Universal Robots PolyScope program: house.urp

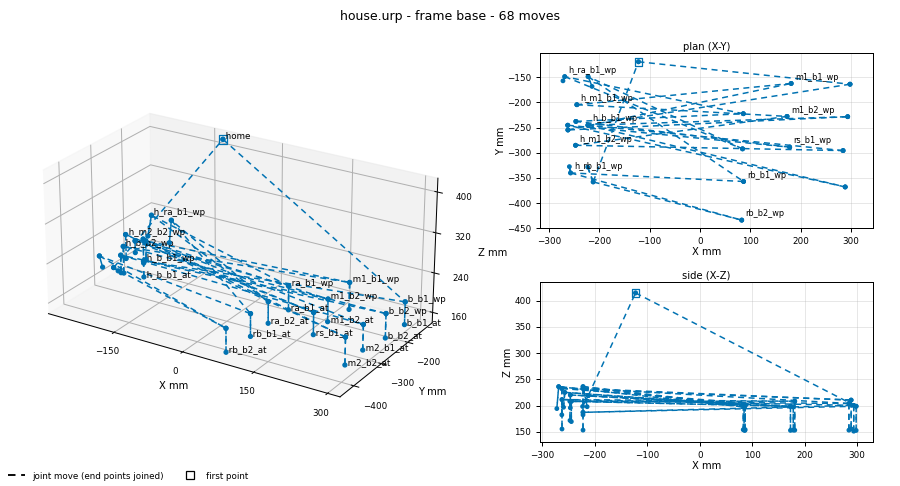
[picture p0: tool path of house.urp in frame base, 68 of 68 moves have a stored position in this frame; points joined in program order, loops and branches not executed]
Program house (installation=default directory=/programs/ITER createdIn=5.3.1.64192 lastSavedIn=5.3.1.64192 robotSerialNumber=20195300365)
Calibrated DH parameters: a=[-0.000093, -0.190649, -0.212673, 0.000091, -0.000205, 0]; d=[0.151591, 44.061648, -42.488068, -1.442789, 0.085322, 0.091911]; alpha=[1.570082, -0.003447, 0.007513, 1.572293, -1.571904, 0]; deltaTheta=[0, -0.672656, 0.728185, -0.055522, 0.000005, 0]
Robot Program (runOnlyOnce=true)
  URCap Gripper Activate (Robotiq_Grippers, Robotiq Inc.) dataModel(ResetAndActivateKey=false)
  URCap Gripper (Robotiq_Grippers, Robotiq Inc.) dataModel(position=50.0, force=100.0, speed=100.0, positionInDouble=50.0, forceInDouble=100.0, speedInDouble=100.0, slaveIds=[9], blocking=true)
  MoveJ speed 60 deg/s, acceleration 80 deg/s^2 (useActiveTCP=true) feature=Base
    Waypoint home: TCP in base x=-122.15 y=-119.32 z=414.454 mm, rx=2.2563 ry=2.1459 rz=-0.0481 rad; joints [-85.681, -56.776, -79.802, -131.025, 89.944, -262.833] deg
  Folder Base
    MoveJ speed 60 deg/s, acceleration 80 deg/s^2 (useActiveTCP=true) feature=Base
      Waypoint b_b1_wp: TCP in base x=297.989 y=-163.874 z=198.695 mm, rx=2.2416 ry=2.1933 rz=-0.0875 rad; joints [-5.657, -99.775, -108.03, -64.017, 87.69, -183.98] deg
      Waypoint b_b1_at: TCP in base x=297.98 y=-163.89 z=152.63 mm, rx=2.2418 ry=2.1932 rz=-0.0874 rad; joints [-5.678, -106.278, -114.473, -51.073, 87.63, -183.927] deg
      URCap Gripper (Robotiq_Grippers, Robotiq Inc.) dataModel(position=100.0, force=100.0, speed=100.0, positionInDouble=100.0, forceInDouble=100.0, speedInDouble=100.0, slaveIds=[9], blocking=true)
      Waypoint b_b1_wp: TCP in base x=297.989 y=-163.874 z=198.695 mm, rx=2.2416 ry=2.1933 rz=-0.0875 rad; joints [-5.657, -99.775, -108.03, -64.017, 87.69, -183.98] deg
      Waypoint h_b_b1_wp: TCP in base x=-222.187 y=-245.349 z=187.06 mm, rx=-3.1315 ry=0.0204 rz=0.0123 rad; joints [-108.957, -99.116, -113.081, -58.146, 89.665, -197.782] deg
      Waypoint h_b_b1_at: TCP in base x=-222.188 y=-245.348 z=153.24 mm, rx=-3.1314 ry=0.0204 rz=0.0122 rad; joints [-108.969, -104.391, -117.643, -48.312, 89.612, -197.745] deg
      URCap Gripper (Robotiq_Grippers, Robotiq Inc.) dataModel(position=50.0, force=100.0, speed=100.0, positionInDouble=50.0, forceInDouble=100.0, speedInDouble=100.0, slaveIds=[9], blocking=true)
      Waypoint h_b_b1_wp: TCP in base x=-222.187 y=-245.349 z=187.06 mm, rx=-3.1315 ry=0.0204 rz=0.0123 rad; joints [-108.957, -99.116, -113.081, -58.146, 89.665, -197.782] deg
    MoveJ speed 60 deg/s, acceleration 80 deg/s^2 (useActiveTCP=true) feature=Base
      Waypoint b_b2_wp: TCP in base x=293.357 y=-228.364 z=200.348 mm, rx=2.2516 ry=2.1757 rz=-0.0473 rad; joints [-17.02, -106.79, -99.111, -64.372, 88.479, -194.689] deg
      Waypoint b_b2_at: TCP in base x=293.371 y=-228.346 z=151.163 mm, rx=2.2516 ry=2.1757 rz=-0.0473 rad; joints [-17.033, -113.072, -105.562, -51.642, 88.423, -194.639] deg
      URCap Gripper (Robotiq_Grippers, Robotiq Inc.) dataModel(position=100.0, force=100.0, speed=100.0, positionInDouble=100.0, forceInDouble=100.0, speedInDouble=100.0, slaveIds=[9], blocking=true)
      Waypoint b_b2_wp: TCP in base x=293.357 y=-228.364 z=200.348 mm, rx=2.2516 ry=2.1757 rz=-0.0473 rad; joints [-17.02, -106.79, -99.111, -64.372, 88.479, -194.689] deg
      Waypoint h_b_b2_wp: TCP in base x=-262.196 y=-254.726 z=211.351 mm, rx=-3.0605 ry=0.0443 rz=-0.0223 rad; joints [-114.749, -105.359, -96.042, -73.109, 89.199, -202.734] deg
      Waypoint h_b_b2_at: TCP in base x=-262.208 y=-254.718 z=155.33 mm, rx=-3.0605 ry=0.0443 rz=-0.0223 rad; joints [-114.774, -111.736, -104.192, -58.581, 89.146, -202.674] deg
      URCap Gripper (Robotiq_Grippers, Robotiq Inc.) dataModel(position=50.0, force=100.0, speed=100.0, positionInDouble=50.0, forceInDouble=100.0, speedInDouble=100.0, slaveIds=[9], blocking=true)
      Waypoint h_b_b2_wp: TCP in base x=-262.196 y=-254.726 z=211.351 mm, rx=-3.0605 ry=0.0443 rz=-0.0223 rad; joints [-114.749, -105.359, -96.042, -73.109, 89.199, -202.734] deg
  Folder Mid_1
    MoveJ speed 60 deg/s, acceleration 80 deg/s^2 (useActiveTCP=true) feature=Base
      Waypoint m1_b1_wp: TCP in base x=181.055 y=-162.39 z=208.274 mm, rx=2.2824 ry=2.1481 rz=-0.0224 rad; joints [-9.334, -71.677, -131.429, -67.006, 89.476, -185.444] deg
      Waypoint m1_b1_at: TCP in base x=181.066 y=-162.388 z=153.109 mm, rx=2.2824 ry=2.1481 rz=-0.0224 rad; joints [-9.367, -82.083, -142.13, -45.899, 89.364, -185.356] deg
      URCap Gripper (Robotiq_Grippers, Robotiq Inc.) dataModel(position=100.0, force=100.0, speed=100.0, positionInDouble=100.0, forceInDouble=100.0, speedInDouble=100.0, slaveIds=[9], blocking=true)
      Waypoint m1_b1_wp: TCP in base x=181.055 y=-162.39 z=208.274 mm, rx=2.2824 ry=2.1481 rz=-0.0224 rad; joints [-9.334, -71.677, -131.429, -67.006, 89.476, -185.444] deg
      Waypoint h_m1_b1_wp: TCP in base x=-244.449 y=-204.582 z=208.1 mm, rx=2.2684 ry=2.1196 rz=0.0229 rad; joints [-116.825, -93.932, -112.747, -63.308, 92.582, -292.535] deg
      Waypoint h_m1_b1_at: TCP in base x=-244.447 y=-204.577 z=169.457 mm, rx=2.2685 ry=2.1196 rz=0.0229 rad; joints [-116.841, -99.299, -118.834, -51.852, 92.525, -292.487] deg
      URCap Gripper (Robotiq_Grippers, Robotiq Inc.) dataModel(position=50.0, force=100.0, speed=100.0, positionInDouble=50.0, forceInDouble=100.0, speedInDouble=100.0, slaveIds=[9], blocking=true)
      Waypoint h_m1_b1_wp: TCP in base x=-244.449 y=-204.582 z=208.1 mm, rx=2.2684 ry=2.1196 rz=0.0229 rad; joints [-116.825, -93.932, -112.747, -63.308, 92.582, -292.535] deg
    MoveJ speed 60 deg/s, acceleration 80 deg/s^2 (useActiveTCP=true) feature=Base
      Waypoint m1_b2_wp: TCP in base x=172.9 y=-227.784 z=198.59 mm, rx=2.2733 ry=2.1297 rz=0.0128 rad; joints [-25.861, -85.885, -124.428, -58.034, 90.195, -201.672] deg
      Waypoint m1_b2_at: TCP in base x=172.893 y=-227.779 z=152.722 mm, rx=2.2733 ry=2.1297 rz=0.0127 rad; joints [-25.879, -94.277, -131.683, -42.391, 90.103, -201.614] deg
      URCap Gripper (Robotiq_Grippers, Robotiq Inc.) dataModel(position=100.0, force=100.0, speed=100.0, positionInDouble=100.0, forceInDouble=100.0, speedInDouble=100.0, slaveIds=[9], blocking=true)
      Waypoint m1_b2_wp: TCP in base x=172.9 y=-227.784 z=198.59 mm, rx=2.2733 ry=2.1297 rz=0.0128 rad; joints [-25.861, -85.885, -124.428, -58.034, 90.195, -201.672] deg
      Waypoint h_m1_b2_wp: TCP in base x=-247.009 y=-285.144 z=208.116 mm, rx=2.2684 ry=2.1195 rz=0.0229 rad; joints [-111.389, -107.719, -95.772, -66.28, 92.556, -287.152] deg
      Waypoint h_m1_b2_at: TCP in base x=-246.994 y=-285.166 z=171.647 mm, rx=2.2684 ry=2.1196 rz=0.0229 rad; joints [-111.399, -111.783, -101.037, -56.949, 92.516, -287.113] deg
      URCap Gripper (Robotiq_Grippers, Robotiq Inc.) dataModel(position=50.0, force=100.0, speed=100.0, positionInDouble=50.0, forceInDouble=100.0, speedInDouble=100.0, slaveIds=[9], blocking=true)
      Waypoint h_m1_b2_wp: TCP in base x=-247.009 y=-285.144 z=208.116 mm, rx=2.2684 ry=2.1195 rz=0.0229 rad; joints [-111.389, -107.719, -95.772, -66.28, 92.556, -287.152] deg
  Folder Mid_2
    MoveJ speed 60 deg/s, acceleration 80 deg/s^2 (useActiveTCP=true) feature=Base
      Waypoint m2_b1_wp: TCP in base x=284.16 y=-295.685 z=203.947 mm, rx=2.2476 ry=2.1381 rz=-0.0269 rad; joints [-27.296, -114.823, -87.386, -65.934, 88.586, -204.141] deg
      Waypoint m2_b1_at: TCP in base x=284.146 y=-295.69 z=153.108 mm, rx=2.2477 ry=2.1381 rz=-0.0269 rad; joints [-27.314, -120.451, -93.885, -53.812, 88.539, -204.094] deg
      URCap Gripper (Robotiq_Grippers, Robotiq Inc.) dataModel(position=100.0, force=100.0, speed=100.0, positionInDouble=100.0, forceInDouble=100.0, speedInDouble=100.0, slaveIds=[9], blocking=true)
      Waypoint m2_b1_wp: TCP in base x=284.16 y=-295.685 z=203.947 mm, rx=2.2476 ry=2.1381 rz=-0.0269 rad; joints [-27.296, -114.823, -87.386, -65.934, 88.586, -204.141] deg
      Waypoint h_m2_b1_wp: TCP in base x=-222.193 y=-245.34 z=232.403 mm, rx=-3.1314 ry=0.0205 rz=0.0123 rad; joints [-108.936, -94.247, -105.13, -70.966, 89.712, -197.837] deg
      Waypoint h_m2_b1_at: TCP in base x=-222.194 y=-245.343 z=182.32 mm, rx=-3.1314 ry=0.0205 rz=0.0122 rad; joints [-108.96, -99.771, -113.792, -56.782, 89.658, -197.776] deg
      URCap Gripper (Robotiq_Grippers, Robotiq Inc.) dataModel(position=50.0, force=100.0, speed=100.0, positionInDouble=50.0, forceInDouble=100.0, speedInDouble=100.0, slaveIds=[9], blocking=true)
      Waypoint h_m2_b1_wp: TCP in base x=-222.193 y=-245.34 z=232.403 mm, rx=-3.1314 ry=0.0205 rz=0.0123 rad; joints [-108.936, -94.247, -105.13, -70.966, 89.712, -197.837] deg
    MoveJ speed 60 deg/s, acceleration 80 deg/s^2 (useActiveTCP=true) feature=Base
      Waypoint m2_b2_wp: TCP in base x=288.413 y=-367.875 z=210.448 mm, rx=2.2648 ry=2.1717 rz=-0.0293 rad; joints [-35.505, -129.071, -61.562, -79.296, 89.186, -212.92] deg
      Waypoint m2_b2_at: TCP in base x=288.4 y=-367.879 z=155.646 mm, rx=2.2649 ry=2.1717 rz=-0.0293 rad; joints [-35.528, -133.111, -69.75, -67.072, 89.162, -212.863] deg
      URCap Gripper (Robotiq_Grippers, Robotiq Inc.) dataModel(position=100.0, force=100.0, speed=100.0, positionInDouble=100.0, forceInDouble=100.0, speedInDouble=100.0, slaveIds=[9], blocking=true)
      Waypoint m2_b2_wp: TCP in base x=288.413 y=-367.875 z=210.448 mm, rx=2.2648 ry=2.1717 rz=-0.0293 rad; joints [-35.505, -129.071, -61.562, -79.296, 89.186, -212.92] deg
      Waypoint h_m2_b2_wp: TCP in base x=-262.568 y=-245.346 z=232.504 mm, rx=-3.1314 ry=0.0205 rz=0.0123 rad; joints [-115.613, -101.169, -97.08, -72.022, 89.654, -204.539] deg
      Waypoint h_m2_b2_at: TCP in base x=-262.563 y=-245.347 z=182.321 mm, rx=-3.1314 ry=0.0204 rz=0.0123 rad; joints [-115.635, -106.202, -105.428, -58.642, 89.608, -204.482] deg
      URCap Gripper (Robotiq_Grippers, Robotiq Inc.) dataModel(position=50.0, force=100.0, speed=100.0, positionInDouble=50.0, forceInDouble=100.0, speedInDouble=100.0, slaveIds=[9], blocking=true)
      Waypoint h_m2_b2_wp: TCP in base x=-262.568 y=-245.346 z=232.504 mm, rx=-3.1314 ry=0.0205 rz=0.0123 rad; joints [-115.613, -101.169, -97.08, -72.022, 89.654, -204.539] deg
  Folder Roof_Support
    MoveJ speed 60 deg/s, acceleration 80 deg/s^2 (useActiveTCP=true) feature=Base
      Waypoint rs_b1_wp: TCP in base x=178.189 y=-288.881 z=197.62 mm, rx=2.2755 ry=2.1482 rz=-0.0598 rad; joints [-35.237, -99.413, -109.73, -60.586, 88.002, -211.537] deg
      Waypoint rs_b1_at: TCP in base x=178.176 y=-288.898 z=153.166 mm, rx=2.2756 ry=2.1481 rz=-0.0597 rad; joints [-35.256, -105.949, -115.836, -47.945, 87.938, -211.491] deg
      URCap Gripper (Robotiq_Grippers, Robotiq Inc.) dataModel(position=100.0, force=100.0, speed=100.0, positionInDouble=100.0, forceInDouble=100.0, speedInDouble=100.0, slaveIds=[9], blocking=true)
      Waypoint rs_b1_wp: TCP in base x=178.189 y=-288.881 z=197.62 mm, rx=2.2755 ry=2.1482 rz=-0.0598 rad; joints [-35.237, -99.413, -109.73, -60.586, 88.002, -211.537] deg
      Waypoint h_rs_b1_wp: TCP in base x=-246.367 y=-237.744 z=220.188 mm, rx=2.2465 ry=2.1469 rz=-0.0526 rad; joints [-114.098, -97.736, -106.012, -63.655, 91.346, -291.09] deg
      Waypoint h_rs_b1_at: TCP in base x=-246.359 y=-237.738 z=195.667 mm, rx=2.2465 ry=2.1469 rz=-0.0525 rad; joints [-114.107, -100.481, -110.105, -56.82, 91.317, -291.061] deg
      URCap Gripper (Robotiq_Grippers, Robotiq Inc.) dataModel(position=50.0, force=100.0, speed=100.0, positionInDouble=50.0, forceInDouble=100.0, speedInDouble=100.0, slaveIds=[9], blocking=true)
      Waypoint h_rs_b1_wp: TCP in base x=-246.367 y=-237.744 z=220.188 mm, rx=2.2465 ry=2.1469 rz=-0.0526 rad; joints [-114.098, -97.736, -106.012, -63.655, 91.346, -291.09] deg
  Folder Roof_A
    MoveJ speed 60 deg/s, acceleration 80 deg/s^2 (useActiveTCP=true) feature=Base
      Waypoint ra_b1_wp: TCP in base x=86.073 y=-222.471 z=201.302 mm, rx=2.2691 ry=2.1657 rz=0.0264 rad; joints [-36.408, -71.347, -133.953, -64.196, 91.272, -213.297] deg
      Waypoint ra_b1_at: TCP in base x=86.083 y=-222.473 z=152.576 mm, rx=2.269 ry=2.1657 rz=0.0264 rad; joints [-36.437, -81.188, -143.371, -44.93, 91.165, -213.22] deg
      URCap Gripper (Robotiq_Grippers, Robotiq Inc.) dataModel(position=100.0, force=100.0, speed=100.0, positionInDouble=100.0, forceInDouble=100.0, speedInDouble=100.0, slaveIds=[9], blocking=true)
      Waypoint ra_b1_wp: TCP in base x=86.073 y=-222.471 z=201.302 mm, rx=2.2691 ry=2.1657 rz=0.0264 rad; joints [-36.408, -71.347, -133.953, -64.196, 91.272, -213.297] deg
      Waypoint h_ra_b1_wp: TCP in base x=-268.55 y=-148.787 z=236.04 mm, rx=2.7608 ry=-0.1306 rz=0.0749 rad; joints [-131.096, -88.368, -118.927, -47.1, 105.838, -213.026] deg
      Waypoint h_ra_b1_at: TCP in base x=-272.048 y=-157.193 z=194.251 mm, rx=2.7928 ry=-0.086 rz=0.1068 rad; joints [-130.55, -96.287, -122.586, -37.872, 105.802, -214.66] deg
      URCap Gripper (Robotiq_Grippers, Robotiq Inc.) dataModel(position=50.0, force=100.0, speed=100.0, positionInDouble=50.0, forceInDouble=100.0, speedInDouble=100.0, slaveIds=[9], blocking=true)
      Waypoint h_ra_b1_wp: TCP in base x=-268.55 y=-148.787 z=236.04 mm, rx=2.7608 ry=-0.1306 rz=0.0749 rad; joints [-131.096, -88.368, -118.927, -47.1, 105.838, -213.026] deg
    MoveJ speed 60 deg/s, acceleration 80 deg/s^2 (useActiveTCP=true) feature=Base
      Waypoint ra_b2_wp: TCP in base x=84.513 y=-292.229 z=197.151 mm, rx=-2.2623 ry=-2.1713 rz=-0.0203 rad; joints [-48.932, -91.406, -118.605, -60.289, 91.026, -226.153] deg
      Waypoint ra_b2_at: TCP in base x=84.516 y=-292.24 z=153.286 mm, rx=-2.2623 ry=-2.1713 rz=-0.0203 rad; joints [-48.95, -98.655, -125.185, -46.457, 90.95, -226.1] deg
      URCap Gripper (Robotiq_Grippers, Robotiq Inc.) dataModel(position=100.0, force=100.0, speed=100.0, positionInDouble=100.0, forceInDouble=100.0, speedInDouble=100.0, slaveIds=[9], blocking=true)
      Waypoint ra_b2_wp: TCP in base x=84.513 y=-292.229 z=197.151 mm, rx=-2.2623 ry=-2.1713 rz=-0.0203 rad; joints [-48.932, -91.406, -118.605, -60.289, 91.026, -226.153] deg
      Waypoint h_ra_b2_wp: TCP in base x=-222.173 y=-148.778 z=236.048 mm, rx=2.7617 ry=-0.0717 rz=0.0011 rad; joints [-121.367, -76.176, -130.557, -44.074, 100.878, -206.047] deg
      Waypoint h_ra_b2_at: TCP in base x=-214.314 y=-168.312 z=197.793 mm, rx=2.8721 ry=-0.0559 rz=-0.0607 rad; joints [-115.061, -82.329, -135.249, -37.27, 94.17, -201.737] deg
      URCap Gripper (Robotiq_Grippers, Robotiq Inc.) dataModel(position=50.0, force=100.0, speed=100.0, positionInDouble=50.0, forceInDouble=100.0, speedInDouble=100.0, slaveIds=[9], blocking=true)
      Waypoint h_ra_b2_wp: TCP in base x=-222.173 y=-148.778 z=236.048 mm, rx=2.7617 ry=-0.0717 rz=0.0011 rad; joints [-121.367, -76.176, -130.557, -44.074, 100.878, -206.047] deg
  Folder Roof_B
    MoveJ speed 60 deg/s, acceleration 80 deg/s^2 (useActiveTCP=true) feature=Base
      Waypoint rb_b1_wp: TCP in base x=86.592 y=-357.042 z=199.917 mm, rx=-2.253 ry=-2.1828 rz=0.0385 rad; joints [-55.332, -105.821, -100.691, -63.448, 88.848, -233.148] deg
      Waypoint rb_b1_at: TCP in base x=86.564 y=-357.044 z=154.241 mm, rx=-2.253 ry=-2.1828 rz=0.0385 rad; joints [-55.35, -111.723, -106.76, -51.481, 88.791, -233.104] deg
      URCap Gripper (Robotiq_Grippers, Robotiq Inc.) dataModel(position=100.0, force=100.0, speed=100.0, positionInDouble=100.0, forceInDouble=100.0, speedInDouble=100.0, slaveIds=[9], blocking=true)
      Waypoint rb_b1_wp: TCP in base x=86.592 y=-357.042 z=199.917 mm, rx=-2.253 ry=-2.1828 rz=0.0385 rad; joints [-55.332, -105.821, -100.691, -63.448, 88.848, -233.148] deg
      Waypoint h_rb_b1_wp: TCP in base x=-256.938 y=-340.018 z=225.107 mm, rx=-2.8953 ry=0.0291 rz=0.0394 rad; joints [-107.997, -121.864, -65.138, -95.964, 84.649, -196.093] deg
      Waypoint h_rb_b1_at: TCP in base x=-259.31 y=-327.534 z=196.716 mm, rx=-2.8001 ry=0.0477 rz=0.0337 rad; joints [-108.564, -122.963, -69.719, -95.569, 83.225, -195.35] deg
      URCap Gripper (Robotiq_Grippers, Robotiq Inc.) dataModel(position=50.0, force=100.0, speed=100.0, positionInDouble=50.0, forceInDouble=100.0, speedInDouble=100.0, slaveIds=[9], blocking=true)
      Waypoint h_rb_b1_wp: TCP in base x=-256.938 y=-340.018 z=225.107 mm, rx=-2.8953 ry=0.0291 rz=0.0394 rad; joints [-107.997, -121.864, -65.138, -95.964, 84.649, -196.093] deg
    MoveJ speed 60 deg/s, acceleration 80 deg/s^2 (useActiveTCP=true) feature=Base
      Waypoint rb_b2_wp: TCP in base x=82.912 y=-433.746 z=201.512 mm, rx=-2.2722 ry=-2.1478 rz=0.0068 rad; joints [-61.956, -123.229, -73.621, -73.849, 89.808, -238.483] deg
      Waypoint rb_b2_at: TCP in base x=82.913 y=-433.742 z=153.995 mm, rx=-2.2723 ry=-2.1477 rz=0.0067 rad; joints [-61.973, -127.536, -80.033, -63.13, 89.779, -238.434] deg
      URCap Gripper (Robotiq_Grippers, Robotiq Inc.) dataModel(position=100.0, force=100.0, speed=100.0, positionInDouble=100.0, forceInDouble=100.0, speedInDouble=100.0, slaveIds=[9], blocking=true)
      Waypoint rb_b2_wp: TCP in base x=82.912 y=-433.746 z=201.512 mm, rx=-2.2722 ry=-2.1478 rz=0.0068 rad; joints [-61.956, -123.229, -73.621, -73.849, 89.808, -238.483] deg
      Waypoint h_rb_b2_wp: TCP in base x=-212.089 y=-357.895 z=218.999 mm, rx=-2.8382 ry=0.0039 rz=0.0883 rad; joints [-100.863, -120.72, -67.712, -97.932, 83.683, -189.646] deg
      Waypoint h_rb_b2_at: TCP in base x=-222.968 y=-328.436 z=198.256 mm, rx=-2.8131 ry=0.0005 rz=0.0189 rad; joints [-103.782, -117.811, -77.473, -92.811, 85.184, -192.786] deg
      URCap Gripper (Robotiq_Grippers, Robotiq Inc.) dataModel(position=50.0, force=100.0, speed=100.0, positionInDouble=50.0, forceInDouble=100.0, speedInDouble=100.0, slaveIds=[9], blocking=true)
      Waypoint h_rb_b2_wp: TCP in base x=-212.089 y=-357.895 z=218.999 mm, rx=-2.8382 ry=0.0039 rz=0.0883 rad; joints [-100.863, -120.72, -67.712, -97.932, 83.683, -189.646] deg
  MoveJ speed 60 deg/s, acceleration 80 deg/s^2 (useActiveTCP=true) feature=Base
    Waypoint home: TCP in base x=-122.15 y=-119.32 z=414.454 mm, rx=2.2563 ry=2.1459 rz=-0.0481 rad; joints [-85.681, -56.776, -79.802, -131.025, 89.944, -262.833] deg
